// SIMATIC S7-200 project (STEP 7-Micro/WIN), CPU 224 REL 02.01

ORGANIZATION_BLOCK 程序块:OB1
TITLE=【PLC收尘器程序实例】
// 操作员通过现场模式开关进入现场模式，或通过中控模式开关切换到中控模式。在现场模式下，按下自启按钮触发系统运行，最终点亮系统运行指示灯并置位系统运行标志；按下自停按钮则停止系统。在中控模式下，中控启停信号通过远程控制置位或复位系统运行标志。
// 系统运行时，自动清灰功能通过脉冲周期定时器每1000个时间单位触发一次，当前处理的室编号递增，分别激活各室脉冲阀和提升阀。当室编号超过7时，它会自动重置为1，形成循环清灰模式。清灰过程中，提升阀延时定时器等待400个时间单位后打开提升阀，脉冲阀在触发后持续运行至脉冲阀延时定时器415个时间单位关闭。为了触发这一过程，脉冲触发定时器每300个时间单位检查一次，仅在系统运行标志或任意室手动触发保持置位时启动。
// 除了自动清灰，系统支持手动操作，操作员可通过按下各室手动触发按钮立即启动对应室的清灰，但仅在脉冲周期定时器未运行时生效，手动触发后对应的手动触发保持置位。
// 若系统检测到异常，报警条件置位时点亮报警指示灯，按下报警复位按钮触发时熄灭。
// 
BEGIN
Network 1 //   I0.2  现场模式            I1.0中控模式
LD     I0.2
AN     I1.0
=      M1.2
?000
Network 2 // I0.0  自启      I0.1 自停  I1.1中控启停
LD     M1.2
LD     I0.0
O      M1.1
ALD
AN     I0.1
=      M1.1
Network 3
// 
// 
LD     M1.1
AN     I1.1
LDN    M1.1
A      I1.0
A      I1.1
OLD
EU
S      M1.0, 1
Network 4
// 
// 
LD     I1.1
O      M1.1
ED
LD     I0.2
EU
LD     I1.0
ED
OLD
OLD
R      M1.0, 1
Network 5
LD     M1.0
=      Q0.0
Network 6 // 网络题目 (单行)
//  
// 网络注释
//  
// 
LD     T101
TON    T33, +1000
TON    T34, +400
TON    T35, +415
ED
INCB   VB100
Network 7
LD     M1.0
O      M2.0
O      M2.1
O      M2.2
O      M2.3
O      M2.4
O      M2.5
O      M2.6
LPS
AN     T33
TON    T101, +300
LPP
AB>    VB100, 7
MOVB   1, VB100
Network 8 // 一室 
// q2.1=1室提升阀，q2.0=1室脉冲阀
// 
LD     T101
AB=    VB100, 1
=      Q2.0
A      T34
AN     T35
=      Q2.1
Network 9 // 二室 
// q2.3=2室提升阀，q2.2=2室脉冲阀。以下顺延。
// 
LD     T101
AB=    VB100, 2
=      Q2.2
A      T34
AN     T35
=      Q2.3
Network 10 // 三室 
// 
// 
LD     T101
AB=    VB100, 3
=      Q2.4
A      T34
AN     T35
=      Q2.5
Network 11 // 四室 
// 
// 
LD     T101
AB=    VB100, 4
=      Q2.6
A      T34
AN     T35
=      Q2.7
Network 12 // 五室 
// 
// 
LD     T101
AB=    VB100, 5
=      Q3.0
A      T34
AN     T35
=      Q3.1
Network 13 // 六室 
// 
// 
LD     T101
AB=    VB100, 6
=      Q3.2
A      T34
AN     T35
=      Q3.3
Network 14 // 七室 
// 
// 
LD     T101
AB=    VB100, 7
=      Q3.4
A      T34
AN     T35
=      Q3.5
Network 15 // 报警信号
// 
// 
LD     SM5.0
S      Q0.1, 1
Network 16
LD     I0.7
R      Q0.1, 1
Network 17
LDN    M1.0
MOVB   0, VB100
Network 18
LDN    T33
LD     I1.2
O      M2.0
ALD
=      M2.0
MOVB   1, VB100
Network 19
LDN    T33
LD     I1.3
O      M2.1
ALD
=      M2.1
MOVB   2, VB100
Network 20
LDN    T33
LD     I1.4
O      M2.2
ALD
=      M2.2
MOVB   3, VB100
Network 21
LDN    T33
LD     I1.5
O      M2.3
ALD
=      M2.3
MOVB   4, VB100
Network 22
LDN    T33
LD     I2.0
O      M2.4
ALD
=      M2.4
MOVB   5, VB100
Network 23
LDN    T33
LD     I2.1
O      M2.5
ALD
=      M2.5
MOVB   6, VB100
Network 24
LDN    T33
LD     I2.2
O      M2.6
ALD
=      M2.6
MOVB   7, VB100
END_ORGANIZATION_BLOCK
